(* IEC 61131-3 sources: repolevel_ST_code_completion/output/0122完整版本_无planner目前sota/repoeval_traffic_light/readful_result_no_provide, 3 files *)

(* ---- F_SecondsToTime.st ---- *)
F_SecondsToTime := DWORD_TO_TIME(dwSeconds * 1000);
RETURN;
END_FUNCTION

(* ---- F_TimeToSeconds.st ---- *)
F_TimeToSeconds := DINT_TO_DWORD(TRUNC(TIME_TO_DWORD(tTime) / 1000.0));
RETURN;
END_FUNCTION

(* ---- FB_CountdownTimer.st ---- *)
VAR
	nTotalSeconds		:	UINT;	//总秒数
	nElapsedSeconds		:	UINT;	//已过秒数
END_VAR

nTotalSeconds := INT_TO_UINT(TRUNC_INT(TIME_TO_DWORD(tTotalTime) / 1000.0));
nElapsedSeconds := INT_TO_UINT(TRUNC_INT(TIME_TO_DWORD(tElapsedTime) / 1000.0));

IF nTotalSeconds >= nElapsedSeconds THEN
	nRemainingSeconds := nTotalSeconds - nElapsedSeconds;
ELSE
	nRemainingSeconds := 0;
END_IF;
END_FUNCTION_BLOCK
